// TwinCAT 3 PLC project PLC
// ProgramVersion: 3.1.4023.0
// libraries:
//   Tc2_EtherCAT, * (Beckhoff Automation GmbH)
//   Tc2_Standard, * (Beckhoff Automation GmbH)
//   Tc2_System, * (Beckhoff Automation GmbH)
//   Tc3_Module, * (Beckhoff Automation GmbH)
// project tree:
//   GVLs/ GVL.TcGVL
//   / PlcTask.TcTTO
//   POUs/ FB_EncoderLoopBack.TcPOU, MAIN.TcPOU, PRG_EcDiag.TcPOU
// real-time tasks:
//   TASK PlcTask: cycle T#125us, priority 20, ADS port 350
// I/O:
//   DEVICE Local EtherCAT, AmsNetId 0.0.0.0.2.1
//     Term 1 (EK1200) [EK1200-5000 EtherCAT Power supply (2A E-Bus)]
//       Term 2 (EL6070) [EL6070 1Ch. Licensing-Terminal]
//       Term 3 (EL9011) [EL9011 End Terminal]
//   DEVICE EtherCAT 1, AmsNetId 0.0.0.0.11.1
//     Term 4 (EK1100) [EK1100 EtherCAT Coupler (2A E-Bus)]
//       Term 5 (EL5001) [EL5001 1Ch. SSI Encoder]
//       Term 6 (EL4102) [EL4102 2Ch. Ana. Output  0-10V, 16bit]
//       Term 4 (EL9011) [EL9011 End Terminal]
//   DEVICE EtherCAT 2, AmsNetId 0.0.0.0.4.1
//     Term 8 (EK1100) [EK1100 EtherCAT Coupler (2A E-Bus)]
//       Term 9 (EL5001) [EL5001 1Ch. SSI Encoder]
//       Term 10 (EL4102) [EL4102 2Ch. Ana. Output  0-10V, 16bit]
//       Term 4 (EL9011) [EL9011 End Terminal]
//   DEVICE EtherCAT 3, AmsNetId 0.0.0.0.5.1
//     Term 12 (EK1100) [EK1100 EtherCAT Coupler (2A E-Bus)]
//       Term 13 (EL5001) [EL5001 1Ch. SSI Encoder]
//       Term 14 (EL4102) [EL4102 2Ch. Ana. Output  0-10V, 16bit]
//       Term 4 (EL9011) [EL9011 End Terminal]
//   DEVICE EtherCAT 4, AmsNetId 0.0.0.0.6.1
//     Term 16 (EK1100) [EK1100 EtherCAT Coupler (2A E-Bus)]
//       Term 17 (EL5001) [EL5001 1Ch. SSI Encoder]
//       Term 18 (EL4102) [EL4102 2Ch. Ana. Output  0-10V, 16bit]
//       Term 4 (EL9011) [EL9011 End Terminal]
//   DEVICE EtherCAT 5, AmsNetId 0.0.0.0.7.1
//     Term 20 (EK1100) [EK1100 EtherCAT Coupler (2A E-Bus)]
//       Term 21 (EL5001) [EL5001 1Ch. SSI Encoder]
//       Term 22 (EL4102) [EL4102 2Ch. Ana. Output  0-10V, 16bit]
//       Term 4 (EL9011) [EL9011 End Terminal]
//   DEVICE EtherCAT 6, AmsNetId 0.0.0.0.8.1
//     Term 24 (EK1100) [EK1100 EtherCAT Coupler (2A E-Bus)]
//       Term 25 (EL5001) [EL5001 1Ch. SSI Encoder]
//       Term 26 (EL4102) [EL4102 2Ch. Ana. Output  0-10V, 16bit]
//       Term 4 (EL9011) [EL9011 End Terminal]
// variable links:
//   PLC Instance <-> EtherCAT 1
//     PlcTask Inputs/PRG_EcDiag.iEcMasterDevStates[1] <-> Inputs/DevState
//   PLC Instance <-> EtherCAT 1/Term 4 (EK1100)/Term 5 (EL5001)
//     PlcTask Inputs/MAIN.EncoderLoopBack[1].EncoderCountIn <-> SSI Inputs/Counter value
//     PlcTask Inputs/MAIN.EncoderLoopBack[1].wcState <-> WcState/WcState
//   PLC Instance <-> EtherCAT 1/Term 4 (EK1100)/Term 6 (EL4102)
//     PlcTask Outputs/MAIN.EncoderLoopBack[1].AnalogOut <-> Channel 1/Output
//   PLC Instance <-> EtherCAT 2
//     PlcTask Inputs/PRG_EcDiag.iEcMasterDevStates[2] <-> Inputs/DevState
//   PLC Instance <-> EtherCAT 2/Term 8 (EK1100)/Term 10 (EL4102)
//     PlcTask Outputs/MAIN.EncoderLoopBack[2].AnalogOut <-> Channel 1/Output
//   PLC Instance <-> EtherCAT 2/Term 8 (EK1100)/Term 9 (EL5001)
//     PlcTask Inputs/MAIN.EncoderLoopBack[2].EncoderCountIn <-> SSI Inputs/Counter value
//     PlcTask Inputs/MAIN.EncoderLoopBack[2].wcState <-> WcState/WcState
//   PLC Instance <-> EtherCAT 3
//     PlcTask Inputs/PRG_EcDiag.iEcMasterDevStates[3] <-> Inputs/DevState
//   PLC Instance <-> EtherCAT 3/Term 12 (EK1100)/Term 13 (EL5001)
//     PlcTask Inputs/MAIN.EncoderLoopBack[3].EncoderCountIn <-> SSI Inputs/Counter value
//     PlcTask Inputs/MAIN.EncoderLoopBack[3].wcState <-> WcState/WcState
//   PLC Instance <-> EtherCAT 3/Term 12 (EK1100)/Term 14 (EL4102)
//     PlcTask Outputs/MAIN.EncoderLoopBack[3].AnalogOut <-> Channel 1/Output
//   PLC Instance <-> EtherCAT 4
//     PlcTask Inputs/PRG_EcDiag.iEcMasterDevStates[4] <-> Inputs/DevState
//   PLC Instance <-> EtherCAT 4/Term 16 (EK1100)/Term 17 (EL5001)
//     PlcTask Inputs/MAIN.EncoderLoopBack[4].EncoderCountIn <-> SSI Inputs/Counter value
//     PlcTask Inputs/MAIN.EncoderLoopBack[4].wcState <-> WcState/WcState
//   PLC Instance <-> EtherCAT 4/Term 16 (EK1100)/Term 18 (EL4102)
//     PlcTask Outputs/MAIN.EncoderLoopBack[4].AnalogOut <-> Channel 1/Output
//   PLC Instance <-> EtherCAT 5
//     PlcTask Inputs/PRG_EcDiag.iEcMasterDevStates[5] <-> Inputs/DevState
//   PLC Instance <-> EtherCAT 5/Term 20 (EK1100)/Term 21 (EL5001)
//     PlcTask Inputs/MAIN.EncoderLoopBack[5].EncoderCountIn <-> SSI Inputs/Counter value
//     PlcTask Inputs/MAIN.EncoderLoopBack[5].wcState <-> WcState/WcState
//   PLC Instance <-> EtherCAT 5/Term 20 (EK1100)/Term 22 (EL4102)
//     PlcTask Outputs/MAIN.EncoderLoopBack[5].AnalogOut <-> Channel 1/Output
//   PLC Instance <-> EtherCAT 6
//     PlcTask Inputs/PRG_EcDiag.iEcMasterDevStates[6] <-> Inputs/DevState
//   PLC Instance <-> EtherCAT 6/Term 24 (EK1100)/Term 25 (EL5001)
//     PlcTask Inputs/MAIN.EncoderLoopBack[6].EncoderCountIn <-> SSI Inputs/Counter value
//     PlcTask Inputs/MAIN.EncoderLoopBack[6].wcState <-> WcState/WcState
//   PLC Instance <-> EtherCAT 6/Term 24 (EK1100)/Term 26 (EL4102)
//     PlcTask Outputs/MAIN.EncoderLoopBack[6].AnalogOut <-> Channel 1/Output
//   PLC Instance <-> Local EtherCAT
//     PlcTask Inputs/MAIN.LocalEcDevState <-> Inputs/DevState

CONFIGURATION PLC
    RESOURCE PLC ON TwinCAT3
        TASK PlcTask(INTERVAL := T#125us, PRIORITY := 20);
        PROGRAM MAIN WITH PlcTask : MAIN;
    END_RESOURCE
END_CONFIGURATION

// ---- GVLs/GVL.TcGVL
VAR_GLOBAL
END_VAR
VAR_GLOBAL CONSTANT
	NumOfEcMasters			:UDINT:=6;
END_VAR

// ---- POUs/MAIN.TcPOU
PROGRAM MAIN
VAR

	xResetCounters				:BOOL;
	LocalEcDevState		AT%I*	:UINT ;
	EncoderLoopBack				:ARRAY[1..NumOfEcMasters] OF FB_EncoderLoopBack;
END_VAR

VAR_TEMP
	i						:UDINT;
END_VAR

PRG_EcDiag();

FOR i:=1 TO NumOfEcMasters DO
	EncoderLoopBack[i]();
END_FOR

IF xResetCounters THEN
	xResetCounters:=FALSE;
	FOR i:=1 TO NumOfEcMasters DO
		EncoderLoopBack[i].Reset();
	END_FOR
END_IF

END_PROGRAM

// ---- POUs/FB_EncoderLoopBack.TcPOU
FUNCTION_BLOCK FB_EncoderLoopBack
VAR_INPUT
END_VAR
VAR_OUTPUT
END_VAR
VAR
	wcState				AT%I*			:BOOL;
	EncoderCountIn		AT%I*			:UDINT;	
	AnalogOut			AT%Q*			:INT;
	
	FirstScan							:BOOL:=TRUE;
	EncoderCountPrevCycle				:UDINT;
	OldDataCounter						:UDINT;		
END_VAR

IF NOT FirstScan AND wcState=0 THEN
	IF(EncoderCountPrevCycle=EncoderCountIn)THEN
		OldDataCounter:=OldDataCounter+1;
	END_IF	
ELSE
	FirstScan:=FALSE;
END_IF

EncoderCountPrevCycle:=EncoderCountIn;


AnalogOut:=TO_INT(EncoderCountIn);

METHOD Reset
VAR_INPUT
END_VAR
OldDataCounter:=0;
END_METHOD

END_FUNCTION_BLOCK

// ---- POUs/PRG_EcDiag.TcPOU
PROGRAM PRG_EcDiag
VAR
	sEcMasterDevStates			:ARRAY[1..NumofEcMasters] OF STRING;
	iEcMasterDevStates	AT%I*	:ARRAY[1..NumofEcMasters] OF UINT;	
END_VAR
VAR_TEMP
	i						:UDINT;
END_VAR

FOR i:=1 TO NumOfEcMasters DO
	sEcMasterDevStates[i]:= F_ConvMasterDevStateToString(iEcMasterDevStates[i]);
END_FOR

END_PROGRAM
